(* IEC 61131-3 sources: cds-text-sync-reference-project/project-view/PLC/PLC Logic/ST_Application/03_Object_POU_ST/01_PROGRAMM, 6 files *)

(* ---- ST_PROGRAMM.st ---- *)
PROGRAM ST_PROGRAMM
VAR_INPUT
	xEnable : BOOL;          // System enable
	xAutoMode : BOOL;        // Control mode: Auto (True) / Manual (False)
	rLevelSetpoint : REAL;   // Filling level setpoint
	rActualLevel : REAL;     // Current level (from sensor)
END_VAR

VAR_OUTPUT
	xPumpActive : BOOL;      // Output: Pump is active
	xLowLevelAlarm : BOOL;   // Output: Low level alarm
	rFlowRate : REAL;        // Current flow rate
END_VAR

VAR
	fbStartupDelay : TON;    // Startup delay timer
	xInternalError : BOOL;   // Internal error flag
	iStep : INT;             // Current algorithm step
	diGlobalStatus : DINT;   // System status (Moved from VAR_IN_OUT as PROGRAM doesn't support them when called by Task)
	iStartCounter : INT;     // Start counter (Moved from VAR_STAT as all variables in PROGRAM VAR are static by nature)
	iLevelStatus : INT;      // Level diagnostic status (from Method)
	xLevelOk : BOOL;         // Level validity flag (from Method)
	diOperatingHours : DINT; // Operating time in hours (via Property)
	xResetHours : BOOL;      // Manual command to reset hours (via Property)
	fbExample : ST_FB;       // Instance of the example Function Block
END_VAR

VAR_TEMP
	rLevelDiff : REAL;       // Temporary variable: level difference (reset every cycle)
END_VAR

VAR RETAIN
	diOperatingSeconds : DINT; // Retain variable: operating time (not reset on power loss)
END_VAR

VAR CONSTANT
	MAX_CAPACITY : REAL := 500.0; // Constant: maximum tank capacity
	MIN_LIMIT : REAL := 10.0;     // Constant: minimum limit threshold
END_VAR

// --- implementation ---

// 0. Use Method to check if level is within safe range (0 to MAX_CAPACITY)
xLevelOk := ST_METHOD(rValue := rActualLevel,
                      rMin := 0.0,
                      rMax := MAX_CAPACITY,
                      iStatusCode => iLevelStatus);

// 1. Calculate level difference in temporary variable.
rLevelDiff := rLevelSetpoint - rActualLevel;
//Modificataion
// 2. Control logic
IF xEnable AND NOT xInternalError THEN

	IF xAutoMode THEN
		// Start pump based on setpoint with hysteresis
		IF rActualLevel < rLevelSetpoint - 5.0 AND NOT xPumpActive THEN
			fbStartupDelay(IN := TRUE, PT := T#2S);
			IF fbStartupDelay.Q THEN
				xPumpActive := TRUE;
				iStartCounter := iStartCounter + 1; // Update counter
			END_IF
		ELSIF rActualLevel >= rLevelSetpoint THEN
			xPumpActive := FALSE;
			fbStartupDelay(IN := FALSE);
		END_IF
	ELSE
		// In manual mode just monitor limits
		xPumpActive := xEnable AND (rActualLevel < MAX_CAPACITY);
	END_IF

ELSE
	xPumpActive := FALSE;
	fbStartupDelay(IN := FALSE);
END_IF

// 3. Alarm handling
xLowLevelAlarm := (rActualLevel < MIN_LIMIT);

// 4. Operating time accumulation (RETAIN)
IF xPumpActive THEN
	diOperatingSeconds := diOperatingSeconds + 1;
END_IF

// 5. Call Action to calculate flow
ST_ACTION();

// 6. Use Property to work with operating hours
diOperatingHours := ST_PROPERTY; // GET: Read hours converted from seconds

IF xResetHours THEN
    ST_PROPERTY := 0;            // SET: Reset seconds by setting property hours to 0
    xResetHours := FALSE;
END_IF

// 7. Status update
IF xLowLevelAlarm THEN
	diGlobalStatus := 999; // Error code
ELSIF xPumpActive THEN
	diGlobalStatus := 100; // Running
ELSE
	diGlobalStatus := 0;   // Standby
END_IF

// 8. Call example Function Block instance
fbExample(xEnable:= TRUE);
fbExample.ST_FB_Action();
fbExample.ST_FB_Method(iValueToAdd:= 1);

ST_Function(rValue:= 10.0, rMin:= 4.0, rMax:= 20.0);

(* ---- ST_PROGRAMM.ST_ACTION.st ---- *)
// This action simulates flow rate calculation based on pump activity
// Ideally called every cycle when pump is active

IF xPumpActive THEN
    // Simple simulation: flow increases until it reaches a nominal value
    IF rFlowRate < 45.5 THEN
        rFlowRate := rFlowRate + 0.5;
    ELSE
        rFlowRate := 45.5; // Nominal flow
    END_IF
ELSE
    // Flow drops when pump is off
    IF rFlowRate > 0.0 THEN
        rFlowRate := rFlowRate - 1.0;
    ELSE
        rFlowRate := 0.0;
    END_IF
END_IF

(* ---- ST_PROGRAMM.ST_METHOD.st ---- *)
METHOD ST_METHOD : BOOL
VAR_INPUT
	rValue : REAL;       // Value to check
	rMin : REAL;         // Minimum limit
	rMax : REAL;         // Maximum limit
END_VAR
VAR_OUTPUT
	iStatusCode : INT;   // 0: OK, 1: Too Low, 2: Too High
END_VAR

// --- implementation ---

// This method checks if a value is within specified bounds

IF rValue < rMin THEN
	iStatusCode := 1;
	ST_METHOD := FALSE;
ELSIF rValue > rMax THEN
	iStatusCode := 2;
	ST_METHOD := FALSE;
ELSE
	iStatusCode := 0;
	ST_METHOD := TRUE;
END_IF

(* ---- ST_PROGRAMM.ST_PROPERTY.Get.st ---- *)
VAR
END_VAR

// --- implementation ---

// Returns operating time in hours
ST_PROPERTY := diOperatingSeconds / 3600;

(* ---- ST_PROGRAMM.ST_PROPERTY.Set.st ---- *)
VAR
END_VAR

// --- implementation ---

// Allows manual override/reset of operating seconds via hours
diOperatingSeconds := ST_PROPERTY * 3600;

(* ---- ST_PROGRAMM_AUX.st ---- *)
PROGRAM ST_PROGRAMM_AUX
VAR
	diTotalHours : DINT;        // Total operating hours read from main program
	xMaintenanceReq : BOOL;    // Maintenance required flag
	iLogCounter : INT;         // Counter for log entries
	xBIT : BOOL;
END_VAR

VAR CONSTANT
	MAINTENANCE_INTERVAL : DINT := 1000; // Maintenance every 1000 hours
END_VAR

// --- implementation ---

// 1. Accessing property of another program (ST_PROGRAMM)
// This is a GET access to the property in ST_PROGRAMM
diTotalHours := ST_PROGRAMM.ST_PROPERTY;

// 2. Logic to determine if maintenance is needed
IF diTotalHours >= MAINTENANCE_INTERVAL THEN
	xMaintenanceReq := TRUE;
ELSE
	xMaintenanceReq := FALSE;
END_IF

// 3. Example of direct variable access between programs.
// Reading a standard variable from ST_PROGRAMM
IF ST_PROGRAMM.xLowLevelAlarm AND iLogCounter < 100 THEN
    iLogCounter := iLogCounter + 1;
    // Here we could call a logging function
END_IF

// 4. Example of writing to another program
// We can reset the hours in the main program via its property
IF xMaintenanceReq AND ST_PROGRAMM.xAutoMode = FALSE THEN
    // Potentially reset hours after maintenance in manual mode
    // ST_PROGRAMM.ST_PROPERTY := 0; // SET access
END_IF

iLogCounter.0 := xBIT;

iLogCounter := BIT_TO_INT(xBIT);
